PROGRAM Stn055_51_Stn512MainMergePrestop
VAR
	
	{attribute 'TcLinkToOSO' := '.iPuckPresent   :=  <0,1,1>TIIB[N72S00 (AL1332)]^N72S03 (AL2341)^TxPDO^input byte 1;
								 .iBufferFull  :=  <0,1,1>TIIB[N72S00 (AL1332)]^N72S03 (AL2341)^TxPDO^input byte 3;
								 .oStopLower   :=  <0,1,5>TIIB[N72S00 (AL1332)]^N72S02 (EX260)^RxPDO^output byte 1'}
	fbConvStop: FB_ConvStop;
	
END_VAR

//  This code instantiates a component that is implimented as a common function block
//    Note that I/O is linked directly to I/O variables inside the named instance

gStn055_51_Stn512MainMergePrestop.ConvRunning := gConsumed_SafetyInterfaceConv.MtrRunning.Enc062Mtr04;

fbConvStop(
	pStn := ADR(gStn055),
	pCmp := ADR(gStn055_51_Stn512MainMergePrestop),
	pUpstreamStop := 0,
	pStateTraceBuffer := ADR(gStn055_StateTraceBuffer),
	pStateTraceFifo := ADR(gStn055_StateTraceFifo),
	pStats := ADR(gStn055_02_Stats));

END_PROGRAM

(* stored: Version 1.1.0.1, ProductVersion 3.1.4024.6
   POU Stn055_51_Stn512MainMergePrestop: Id {2d33e6fb-0aa3-46c4-8418-286c94454fbb}, SpecialFunc None *)
